// TIA Portal V19 export
FUNCTION_BLOCK "LAF_Checksum"   // FB40, LAD
TITLE = LAF_Checksum / PLC checksum mit ProDiag
AUTHOR : Siemens Digital Industries
FAMILY : LAF
VERSION : 1.2
// The block reads the checksums for PLC standard blocks, for PLC safety blocks and for PLC text lists. The current checksums are compared with the previous values / old values. For each deviation a ProDiag warning is issued, and the colors of the WinCC buttons "Checksum"(SubMenu), "Ok Checksum" and "Settings" (Main Menu) are animated.
// 
// **PLC-Data types**  
// * LAF_typeChecksum  
// * LAF_typeChecksumCatBool  
// * LAF_typeChecksumCatWord  
// 
// **WinCC Screen**  
// 
// {.pageWidth}
// ![Image](LAF_Checksum_PrD/en/image1.PNG)
// 
// **Block call example**  
// {.pageWidth}
// ![Image](LAF_Checksum_PrD/en/image2.PNG)
// The call is shown as “Ladder Diagram” (LAD). 
// 
// **Call interface**  
// The block is called once in the cyclic program. The call takes place in the software unit CentralFunctions -> 05_Diagnostic-> [CallDiagnostic](../Functions/CallDiagnostic.htm)  
// 
// **Internally used “extended instructions / blocks”**  
// GetChecksum, HTA, S_COMP, S_MOVE  
// 
// **Parameters**  
// This block is provided with “pre-defined actual parameters” for structured data types, user constants, system constants etc. Therefor these parameters must be modified only slightly or not at all, if the symbols of DBs, user constants, and system constants have not been changed.
// Der Baustein liest die Checksummen für Standard- und Safety-Bausteine, sowie für Textlisten aus. Die aktuell ausgelesenen Checksummen werden mit den vorherigen Werten (Altwerte) verglichen. Bei Abweichungen wird jeweils eine ProDiag Warnmeldung ausgegeben und die WinCC-Objekte in dem Bild „System & Einstellungen“ farblich animiert. Das Bild ist erreichbar über den Button „System“ (aus jedem Bild, rechts unten).  
// * LSicar_Checksum_PrD:	mit ProDiag-Meldeverfahren 
// * LSicar_Checksum		mit program_Alarm Meldeverfahren
// 
// **PLC-Datentypen**  
//  LSicar_typeChecksum  
//  LSicar_typeChecksumCatBool  
//  LSicar_typeChecksumCatWord  
//  LSicar_typeAlarmText  
//  
// 
// **WinCC-Bild**  
// 
// {.pageWidth}
// ![Image](LSicar_Checksum_PrD/de/image1.PNG)
// 
// **Beispielaufruf**  
// Abbildung in Kontaktplan (KOP), ohne Parameterbeschaltung. D:\Software\Symbols_Icons\BMPs-JPGs-PNGs\Verschiedene\symb_user_goto_transparent.pngEin lauffähiger Programm-Aufruf hierzu ist im „SICAR-StartUp“-Projekt enthalten, incl. der notwendigen HMI-Variablen zur Darstellung der Werte auf dem HMI.  
// 
// **Aufrufschnittstelle**  
// Der Baustein wird einmalig im zyklischen Programm aufgerufen.  
// 
// **Intern verwendete „Erweiterte Anweisungen / Bausteine“**  
// GetChecksum, HTA, S_COMP, S_MOVE  
// 
// **Parameter**
//   
// ![Icon](_Icon/information.PNG) 
// 
// Der Baustein ist mit "Vordefinierten Aktualparametern" versehen für Strukturvariablen, Anwender- und Systemkonstanten etc., die dadurch nicht oder nur geringfügig angepasst werden müssen, vorausgesetzt die Symbolischen Namen von DBs, Anwender-/Systemkonstanten etc. wurden nicht geändert. Die Anpassungen sind notwendig beim Index [i], z.B. für den BA-Bereich oder die HMI-/Panelnummer.  
// 
// * Der Index ist vorbesetzt mit dem Wert [0]. Damit wird auf den Index 0 (Dummy) verwiesen. Sofern der Baustein-Parameter nicht benötigt wird, sind keine Anpassungen notwendig, andernfalls muss der Indexwert angepasst werden.  
// oder  
// * Der Index ist vorbesetzt mit [???]. Dies führt dazu, dass der Aktualparameter beim Bausteinaufruf rot markiert wird; um darauf aufmerksam zu machen, dass der Indexwert des Aktualparameters angepasst werden muss!
// stored: Access Published, IsIECCheckEnabled true, MemoryReserve 100, SetENOAutomatically true
   VAR_INPUT
      plantIdentifier { ExternalAccessible := 'False'; ExternalVisible := 'False'; ExternalWritable := 'False'} : WString[#MAX_CHAR];   // Betriebsmittel Kennzeichen. An diesem Parameter kann ein Text mit max. 24 Zeichen parametriert werden; dies kann beispielweise die Betriebsmittelkennzeichnung sein. Der Wert wird in die ProDiag-Warnmeldung mit eingebracht. / Equipment identifying symbol. The symbol is limited to 24 characters. It can contain the Equipment identifying symbol according to the hardware diagrams. The text assigned here is used for the ProDiag alarm text in the alarm view.
      textListId { ExternalAccessible := 'False'; ExternalVisible := 'False'; ExternalWritable := 'False'} : Int;   // Text list ID
      dateTime { ExternalAccessible := 'False'; ExternalVisible := 'False'; ExternalWritable := 'False'} : Date_And_Time;   // Wird ein Unterschied zwischen der aktuellen und der vorherigen (alten) Checksumme festgestellt, so wird das mit Datum & Uhrzeit abgespeichert und im Bild „Checksumme“ angezeigt. Der Parameter ist vordefiniert und verweist auf nachfolgende Quelle / If the current checksum deviates from the old checksum, date and time are saved and displayed in the screen “Checksum”.
      readChecksum { ExternalAccessible := 'False'; ExternalVisible := 'False'; ExternalWritable := 'False'} : Bool;   // Verwenden Sie hier ein Signal, mit dem die PLC-Checksumme gelesen wird. Es reicht ein Impuls aus. / Assign a signal to read the PLC checksums. A pulse is enough.
      ack { ExternalAccessible := 'False'; ExternalVisible := 'False'; ExternalWritable := 'False'} : Bool;   // Signal mit dem die ProDiag-Warnmeldung quittiert werden kann. Der Parameter ist vordefiniert und verweist auf nachfolgende Quelle. Hinweis: Mit dem globalAck. werden alle anstehenden Meldungen quittiert. Sollen nur die Meldungen für die PLC-Checksumme quittiert werden, so verwenden Sie den Button [OK Checksum] im Bild „Checksum“, siehe WinCC-Bild / For this parameter, assign a signal to reset the ProDiag warnings. Note: All present alarms are reset with the globalAck. If you want to reset only the warnings for the PLC checksums, use the button [OK Checksum] in screen “Checksum".
      hideMessageStandard { ExternalAccessible := 'False'; ExternalVisible := 'False'; ExternalWritable := 'False'} : Bool;   // Der Parameter ist vordefiniert und verweist auf nachfolgende Quelle / The ProDiag warning is suppressed / hidden if a TRUE-Signal is assigned. Note: A TRUE signal does not suppress the color animation of the faceplate and of the WinCC objects in screen “Checksum”. This ensures that the difference of the PLC checksums is visible even if the ProDiag warning is hidden.
      hideMessageSafety { ExternalAccessible := 'False'; ExternalVisible := 'False'; ExternalWritable := 'False'} : Bool;   // Wie bei Parameter „hideMessageStandard“ / Like parameter “hideMessageStandard”
      hideMessageTextlist { ExternalAccessible := 'False'; ExternalVisible := 'False'; ExternalWritable := 'False'} : Bool;   // Wie bei Parameter „hideMessageStandard“ / Like parameter “hideMessageStandard”
   END_VAR
   VAR_OUTPUT
      generalMessage { ExternalAccessible := 'False'; ExternalVisible := 'False'; ExternalWritable := 'False'} : Bool;   // Sammelwarnung / General alarm
   END_VAR
   VAR_IN_OUT
      checksumHmi : "LAF_typeChecksum";   // Transfer of the information for display on the HMI. / PLC checksum for HMI
   END_VAR
   VAR
      statReadChecksumStorage { ExternalAccessible := 'False'; ExternalVisible := 'False'; ExternalWritable := 'False'} : Bool;   // Start: Lesen der PLC Checksummen (Storage) / Start: Read PLC checksum (storage)
      statChecksumStandard { ExternalAccessible := 'False'; ExternalVisible := 'False'; ExternalWritable := 'False'} : Array[0..7] of Byte;   // Checksumme Standard / Checksum Standard
      statChecksumStafety { ExternalAccessible := 'False'; ExternalVisible := 'False'; ExternalWritable := 'False'} : Array[0..7] of Byte;   // Checksumme Safety / Checksum Safety
      statChecksumTextlists { ExternalAccessible := 'False'; ExternalVisible := 'False'; ExternalWritable := 'False'} : Array[0..7] of Byte;   // Checksumme Textlisten / Checksumme Textlists
      statChecksumStandOldNull { ExternalAccessible := 'False'; ExternalVisible := 'False'; ExternalWritable := 'False'} : Bool;   // Vorherige Checksumme = Null (nichts) / Checksum old = null (nothing)
      statChecksumSafeOldNull { ExternalAccessible := 'False'; ExternalVisible := 'False'; ExternalWritable := 'False'} : Bool;   // Vorherige Checksumme = Null (nichts) / Checksum old = null (nothing)
      statChecksumTextlOldNull { ExternalAccessible := 'False'; ExternalVisible := 'False'; ExternalWritable := 'False'} : Bool;   // Vorherige Checksumme = Null (nichts) / Checksum old = null (nothing)
      statChecksumStandDiff { ExternalAccessible := 'False'; ExternalVisible := 'False'; ExternalWritable := 'False'} : Bool;   // Checksumme unterschiedlich Standard / Checksum different Standard
      statChecksumSafeDiff { ExternalAccessible := 'False'; ExternalVisible := 'False'; ExternalWritable := 'False'} : Bool;   // Checksumme unterschiedlich Safety / Checksum different Safety
      statChecksumTextlDiff { ExternalAccessible := 'False'; ExternalVisible := 'False'; ExternalWritable := 'False'} : Bool;   // Checksumme unterschiedlich Textlisten / Checksum different Textlists
      instGetChecksum1 { ExternalAccessible := 'False'; ExternalVisible := 'False'; ExternalWritable := 'False'} : GetChecksum;   // GetChecksum1
      instGetChecksum2 { ExternalAccessible := 'False'; ExternalVisible := 'False'; ExternalWritable := 'False'} : GetChecksum;   // GetChecksum2
      instGetChecksum3 { ExternalAccessible := 'False'; ExternalVisible := 'False'; ExternalWritable := 'False'} : GetChecksum;   // GetChecksum3
      statRetValHta { ExternalAccessible := 'False'; ExternalVisible := 'False'; ExternalWritable := 'False'} : "LAF_typeChecksumCatWord";   // Ret_VAT von HTA / RET_VAL of HTA
      statRisEdgeDiff { ExternalAccessible := 'False'; ExternalVisible := 'False'; ExternalWritable := 'False'} : "LAF_typeChecksumCatBool";   // Steigende Flanke / Rising edge
      statMessageStandModified { ExternalAccessible := 'False'; ExternalVisible := 'False'; ExternalWritable := 'False'} : Bool;   // Meldung: Standard Bausteine wurden modifiziert / Message: Standard blocks are modified
      statMessageSafeModified { ExternalAccessible := 'False'; ExternalVisible := 'False'; ExternalWritable := 'False'} : Bool;   // Meldung: Safety Bausteine wurden modifiziert / Message: Safety blocks are modified
      statMessageTextlModified { ExternalAccessible := 'False'; ExternalVisible := 'False'; ExternalWritable := 'False'} : Bool;   // Meldung: Textlisten wurden modifiziert / Message: Textlists are modified
      statWarnNoStandard { ExternalAccessible := 'False'; ExternalVisible := 'False'; ExternalWritable := 'False'} : UInt;   // Warn Nummer - Standard / Warn number - Standard
      statWarnNoSafety { ExternalAccessible := 'False'; ExternalVisible := 'False'; ExternalWritable := 'False'} : UInt;   // Warn Nummer - Safety / Warn number - Safety
      statWarnNoTextlist { ExternalAccessible := 'False'; ExternalVisible := 'False'; ExternalWritable := 'False'} : UInt;   // Warn Nummer - Textlisten / Warn number - Textlists
   END_VAR
   VAR CONSTANT
      MAX_CHAR : DInt := 24;   // Konstante für Zeichenlänge plantidentifier / Constant length plantidentifier
   END_VAR
   VAR_TEMP   // added for the SCL form of the ladder/FBD networks
      _w1 : Bool;
      _w2 : Bool;
      _w3 : Bool;
   END_VAR
BEGIN

REGION Network 1: Header Info / Änderungshistorie
   // SIEMENS AG / (c)Copyright 2024
   // ------------------------------------------------------------------------------
   // Title:            LAF_InterfaceSignalsBool
   // Comment/Function: The block reads the checksums for PLC standard blocks, for PLC safety blocks and for PLC text lists. The current checksums are compared with the previous values / old values
   // Library/Family:   Library of Automation Framework
   // Author:                Siemens Digital Industry
   // Tested with:       S7-PLCSIM Advanced 6.0
   // Engineering:      TIA Portal V19
   // Restrictions:       ---
   // Requirements:   ---
   // ------------------------------------------------------------------------------
   // Change log table:
   // Version | Date | Expert in charge | Changes applied
   // -------|---------|-------------|--------------------------------------------
   // 01.02.00 | 30.09.2024 | SIMATIC Systems Support | First released version
   // Die Änderungshistorie wird nur in englischer Editiersprache geführt.
END_REGION

REGION Network 2: Description / Beschreibung
   // **Operation mode Automatic / Manual**  
   // The block is independent of operation modes. Therefor it is not assigned to any operation mode area.  
   // 
   // **Alarms**  
   // Alarm texts are stored in the PLC alarm text lists of the software unit GlobalData. This messages are used with proDiag and also in the program alarm version of the block.  
   // 
   // | **No.** | **Message**             |
   // |---------|-------------------------|
   // | 1       | Standard block modified |
   // | 2       | Safety block modified   |
   // | 3       | Textlist modified       |
   // | 4       | Spare4_en               |
   // | 5       | Spare5_en               |
   // | 6       | Spare6_en               |
   // | 7       | Spare7_en               |
   // | 8       | Spare8_en               |
   // 
   // ---
   // 
   // #### PLC Data types 
   // * [LAF_typeChecksum](../Library%20Types/LAF_typeChecksum.htm)  
   // * [LAF_typeChecksumCatBool](../Library%20Types/LAF_typeChecksumCatBool.htm)  
   // * [LAF_typeChecksumCatWord](../Library%20Types/LAF_typeChecksumCatWord.htm)  
   // 
   // 
   // #### WinCC Objects 
   // 
   // **WinCC Screen**  
   // The screen is to be found in the project in the HMI part, in folder “Screens” -> 11_Settings. It consists of several WinCC objects and contains the information shown below.  
   // ![Image](LAF_Checksum_PrD/en/image1.PNG)
   // 
   // ---
   // 
   // #### Further information 
   // 
   // #### Update info
   // 
   // #### Further documentation
   // **Betriebsart Automatik / Hand**  
   // Der Baustein ist keiner Betriebsart / Betriebsartenbereich zugeordnet.  
   // 
   // **Alarme**  
   // Der Baustein generiert die in der PLC-Meldetextliste „PLC_Checksum_PD“ angegebenen Texte als ProDiag-Warnmeldungen, wenn die aktuelle und vorherige (Altwert) Checksumme unterschiedlich sind.  
   // 
   // 
   // Die Textliste „PLC_Checksum_PD“ ist in der PLC-Meldetextliste „GLOBAL_GENERAL_AlarmTextList“ als Eintragsnummer 22 hinterlegt. Siehe auch FB-Parameter: „globalAlarmTextListItem“  
   //  
   // ![Image](LSicar_Checksum_PrD/de/image2.PNG)
   // 
   //  
   // #### PLC Data types 
   // 
   // “_typeChecksum” enthält alle Informationen, die in der Visualisierung angezeigt werden.   
   // 
   // ![Image](LSicar_Checksum_PrD/de/image3.PNG)
   //  
   // “_typeChecksumCatBool” enthält die Struktur für Flankenauswertungen  
   // 
   // ![Image](LSicar_Checksum_PrD/de/image4.PNG)
   //  
   // “_typeChecksumCatWord” enthält die Struktur für RetVal Werte.  
   // 
   // ![Image](LSicar_Checksum_PrD/de/image5.PNG)
   // 
   // Weitere PLC-Datentypen:  
   // 
   // ![Icon](_Icon/reference.PNG)
   // 
   // Siehe LSicar_typeAlarmText.pdf 
   //  
   // 
   // #### WinCC-Bildobjekte
   // 
   // **WinCC-Bild**  
   // Das Bild befindet sich im Projekt im HMI-Teil unter „Bilder“. Es ist erstellt aus mehreren einzelnen WinCC-Objekten und enthält die dargestellten Informationen.  
   // 
   // ![Image](LSicar_Checksum_PrD/de/image6.PNG)
   // 
   // **WinCC-Bildbaustein**  
   // Der Bildbaustein PLC_Checksum befindet sich in der Projektbilbliothek und besteht aus mehreren einzelnen WinCC-Objekten. Er ist in den Startup-Projekten zusätzlich in der Kopfzeile projektiert. Bei Ungleichheit der PLC-Checksummen wird er orange animiert.  
   // In dessen Schnittstelle können Sie die Default-Farbe einstellen. Für das Schnittstellensignal zum Animieren verwenden Sie die HMI-Variable  .summaryModified“.  
   // 
   // ![Image](LSicar_Checksum_PrD/de/image7.PNG)
   // 
   // 
   // #### Further information 
   // 
   // #### Update info
   // 
   // #### Further documentation
END_REGION

REGION Network 3: Call "GetChecksum" and convert to string / Aufruf "GetChecksum" und wandeln in String
   // Read out checksum and convert it to string / Lesen der Prüfsumme und umwandeln in eine Stringvariable
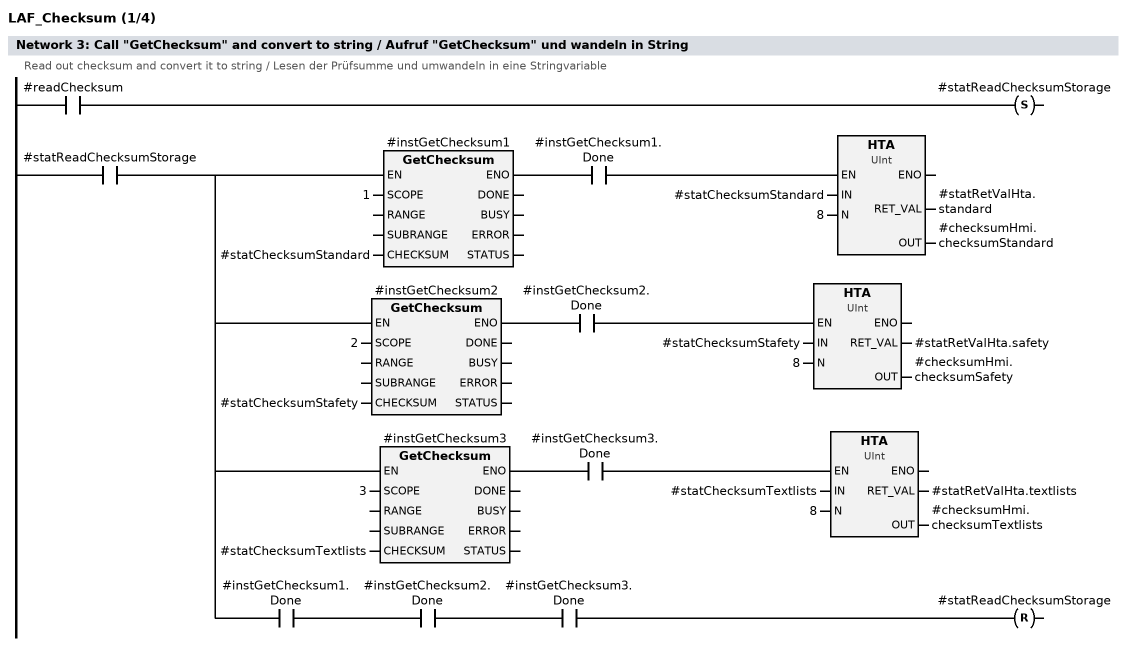
   RUNG wire#powerrail
      Contact( #readChecksum )
      S_Coil( #statReadChecksumStorage )
   END_RUNG
   RUNG wire#powerrail
      Contact( #statReadChecksumStorage )
      wire#w1
      #instGetChecksum1.GetChecksum(Scope := 1, Range :=, Subrange :=, Checksum := #statChecksumStandard, Done =>, Busy =>, Error =>, Status =>)
      Contact( #instGetChecksum1.Done )
      { S7_Templates := "[card := 1, n_type := UInt, in_out_type := Variant]" } HTA(IN := #statChecksumStandard, N := 8, RET_VAL => #statRetValHta.standard, OUT => #checksumHmi.checksumStandard)
   END_RUNG
   RUNG wire#w1
      #instGetChecksum2.GetChecksum(Scope := 2, Range :=, Subrange :=, Checksum := #statChecksumStafety, Done =>, Busy =>, Error =>, Status =>)
      Contact( #instGetChecksum2.Done )
      { S7_Templates := "[card := 1, n_type := UInt, in_out_type := Variant]" } HTA(IN := #statChecksumStafety, N := 8, RET_VAL => #statRetValHta.safety, OUT => #checksumHmi.checksumSafety)
   END_RUNG
   RUNG wire#w1
      #instGetChecksum3.GetChecksum(Scope := 3, Range :=, Subrange :=, Checksum := #statChecksumTextlists, Done =>, Busy =>, Error =>, Status =>)
      Contact( #instGetChecksum3.Done )
      { S7_Templates := "[card := 1, n_type := UInt, in_out_type := Variant]" } HTA(IN := #statChecksumTextlists, N := 8, RET_VAL => #statRetValHta.textlists, OUT => #checksumHmi.checksumTextlists)
   END_RUNG
   RUNG wire#w1
      Contact( #instGetChecksum1.Done )
      Contact( #instGetChecksum2.Done )
      Contact( #instGetChecksum3.Done )
      R_Coil( #statReadChecksumStorage )
   END_RUNG
   // the same network as SCL:
   IF #readChecksum THEN #statReadChecksumStorage := TRUE; END_IF;
   #instGetChecksum1(EN := #statReadChecksumStorage, Scope := 1, Checksum := #statChecksumStandard, ENO => #_w1);   // GetChecksum
   IF #_w1 AND #instGetChecksum1.Done THEN
       #statRetValHta.standard := HTA(IN := #statChecksumStandard, N := 8, OUT => #checksumHmi.checksumStandard);
   END_IF;
   #instGetChecksum2(EN := #statReadChecksumStorage, Scope := 2, Checksum := #statChecksumStafety, ENO => #_w2);   // GetChecksum
   IF #_w2 AND #instGetChecksum2.Done THEN
       #statRetValHta.safety := HTA(IN := #statChecksumStafety, N := 8, OUT => #checksumHmi.checksumSafety);
   END_IF;
   #instGetChecksum3(EN := #statReadChecksumStorage,   // GetChecksum
                     Scope := 3,
                     Checksum := #statChecksumTextlists,
                     ENO => #_w3);
   IF #_w3 AND #instGetChecksum3.Done THEN
       #statRetValHta.textlists := HTA(IN := #statChecksumTextlists, N := 8, OUT => #checksumHmi.checksumTextlists);
   END_IF;
   IF #statReadChecksumStorage AND #instGetChecksum1.Done AND #instGetChecksum2.Done AND #instGetChecksum3.Done THEN
       #statReadChecksumStorage := FALSE;
   END_IF;
END_REGION

REGION Network 4: Overwrite value-before with current-value / Vorheriger Wert mit aktuellem Wert beschreiben
   // Describe old value with current value if old value is still empty (eg. at restart) or if it has been acknowledged with ACK or #HMI.Update_Values_Old / Altwert mit aktuellem Wert beschreiben, falls Altwert noch leer (z.B. bei Neustart) oder wenn Quittiert wurde mit QUIT oder #HMI.Update_Values_Old
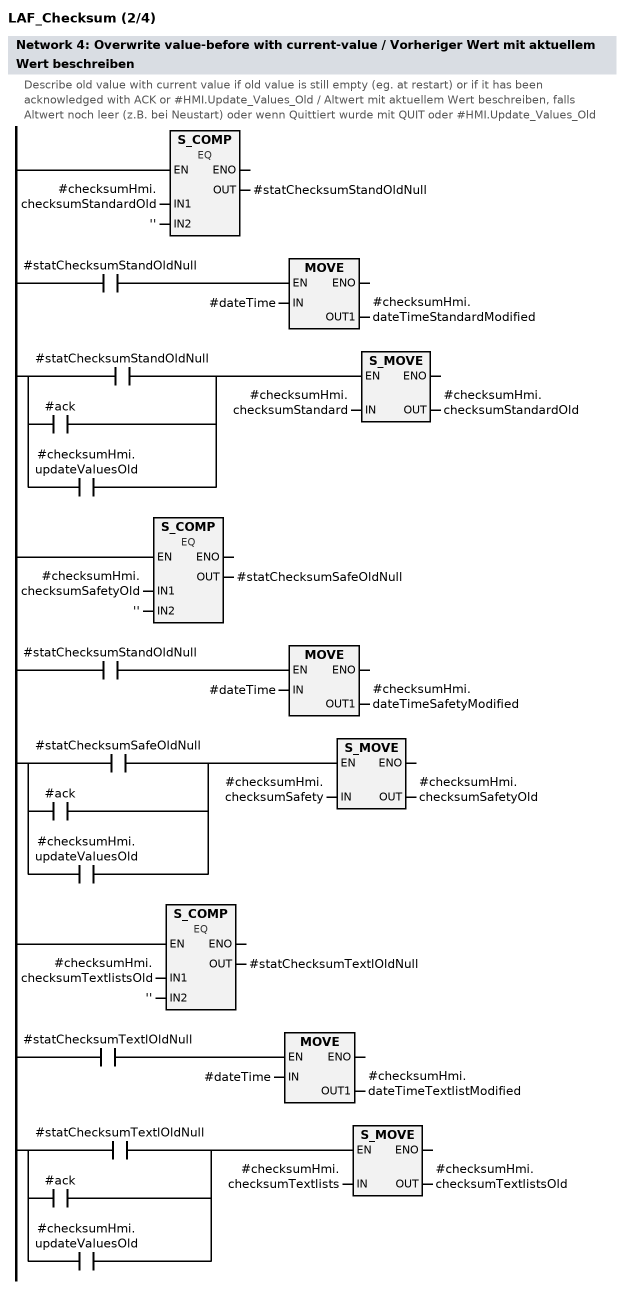
   RUNG wire#powerrail
      { S7_Templates := "[relation := EQ, src_type := String]" } S_COMP(IN1 := #checksumHmi.checksumStandardOld, IN2 := '', OUT => #statChecksumStandOldNull)
   END_RUNG
   RUNG wire#powerrail
      Contact( #statChecksumStandOldNull )
      Move(in := #dateTime, out1 => #checksumHmi.dateTimeStandardModified)
   END_RUNG
   RUNG wire#powerrail
      Contact( #statChecksumStandOldNull )
      wire#w1
      S_Move(in := #checksumHmi.checksumStandard, out => #checksumHmi.checksumStandardOld)
   END_RUNG
   RUNG wire#powerrail
      Contact( #ack )
   END_RUNG wire#w1
   RUNG wire#powerrail
      Contact( #checksumHmi.updateValuesOld )
   END_RUNG wire#w1
   RUNG wire#powerrail
      { S7_Templates := "[relation := EQ, src_type := String]" } S_COMP(IN1 := #checksumHmi.checksumSafetyOld, IN2 := '', OUT => #statChecksumSafeOldNull)
   END_RUNG
   RUNG wire#powerrail
      Contact( #statChecksumStandOldNull )
      Move(in := #dateTime, out1 => #checksumHmi.dateTimeSafetyModified)
   END_RUNG
   RUNG wire#powerrail
      Contact( #statChecksumSafeOldNull )
      wire#w2
      S_Move(in := #checksumHmi.checksumSafety, out => #checksumHmi.checksumSafetyOld)
   END_RUNG
   RUNG wire#powerrail
      Contact( #ack )
   END_RUNG wire#w2
   RUNG wire#powerrail
      Contact( #checksumHmi.updateValuesOld )
   END_RUNG wire#w2
   RUNG wire#powerrail
      { S7_Templates := "[relation := EQ, src_type := String]" } S_COMP(IN1 := #checksumHmi.checksumTextlistsOld, IN2 := '', OUT => #statChecksumTextlOldNull)
   END_RUNG
   RUNG wire#powerrail
      Contact( #statChecksumTextlOldNull )
      Move(in := #dateTime, out1 => #checksumHmi.dateTimeTextlistModified)
   END_RUNG
   RUNG wire#powerrail
      Contact( #statChecksumTextlOldNull )
      wire#w3
      S_Move(in := #checksumHmi.checksumTextlists, out => #checksumHmi.checksumTextlistsOld)
   END_RUNG
   RUNG wire#powerrail
      Contact( #ack )
   END_RUNG wire#w3
   RUNG wire#powerrail
      Contact( #checksumHmi.updateValuesOld )
   END_RUNG wire#w3
   // the same network as SCL:
   S_COMP(IN1 := #checksumHmi.checksumStandardOld, IN2 := '', OUT => #statChecksumStandOldNull);
   IF #statChecksumStandOldNull THEN #checksumHmi.dateTimeStandardModified := #dateTime; END_IF;
   IF #statChecksumStandOldNull OR #ack OR #checksumHmi.updateValuesOld THEN
       #checksumHmi.checksumStandardOld := #checksumHmi.checksumStandard;
   END_IF;
   S_COMP(IN1 := #checksumHmi.checksumSafetyOld, IN2 := '', OUT => #statChecksumSafeOldNull);
   IF #statChecksumStandOldNull THEN #checksumHmi.dateTimeSafetyModified := #dateTime; END_IF;
   IF #statChecksumSafeOldNull OR #ack OR #checksumHmi.updateValuesOld THEN
       #checksumHmi.checksumSafetyOld := #checksumHmi.checksumSafety;
   END_IF;
   S_COMP(IN1 := #checksumHmi.checksumTextlistsOld, IN2 := '', OUT => #statChecksumTextlOldNull);
   IF #statChecksumTextlOldNull THEN #checksumHmi.dateTimeTextlistModified := #dateTime; END_IF;
   IF #statChecksumTextlOldNull OR #ack OR #checksumHmi.updateValuesOld THEN
       #checksumHmi.checksumTextlistsOld := #checksumHmi.checksumTextlists;
   END_IF;
END_REGION

REGION Network 5: Message: Standard blocks are modified / Meldung: Standard Bausteine wurden modifiziert
   // Generate ProDiag message only if it is not deselected (HIDE ... = 0)
   // In the screen always mark the difference in color, by #HMI ... Modified
   // ProDiag-Meldung nur generieren, wenn sie nicht abgewählt ist (HIDE... = 0)
   // Im Bild den Unterschied immer farblich markieren, durch #HMI...Modified
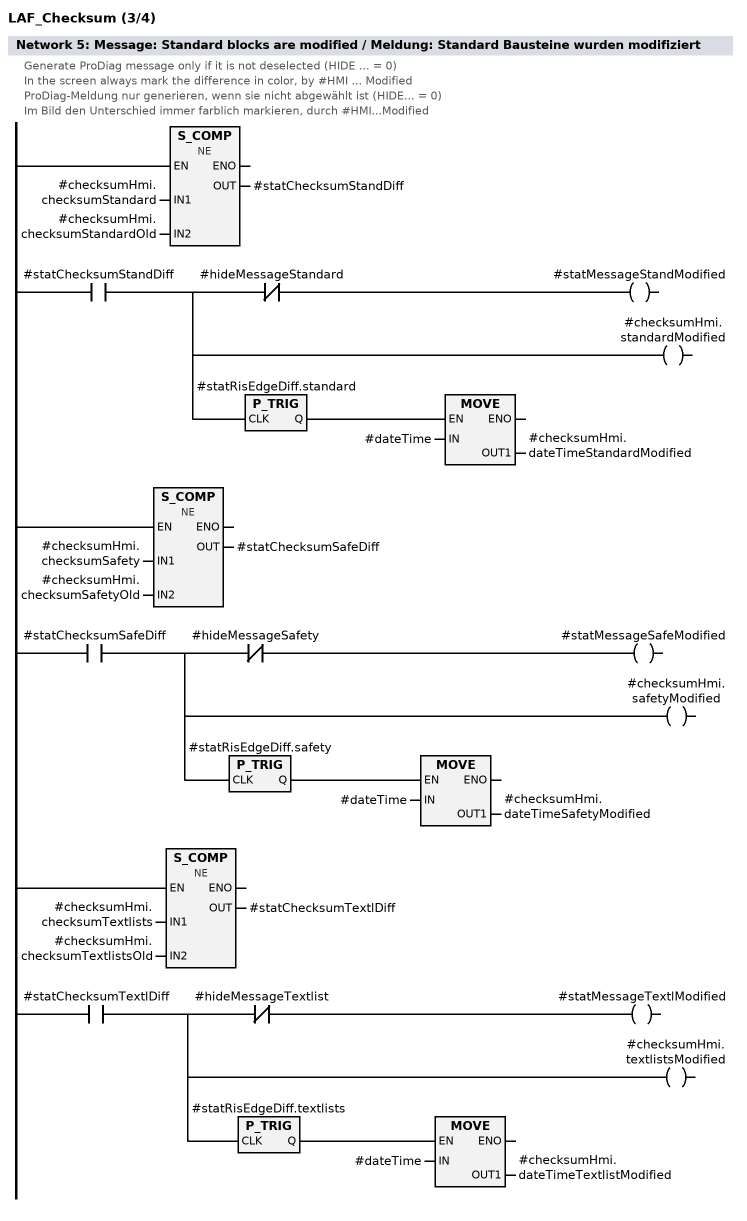
   RUNG wire#powerrail
      { S7_Templates := "[relation := NE, src_type := String]" } S_COMP(IN1 := #checksumHmi.checksumStandard, IN2 := #checksumHmi.checksumStandardOld, OUT => #statChecksumStandDiff)
   END_RUNG
   RUNG wire#powerrail
      Contact( #statChecksumStandDiff )
      wire#w1
      I_Contact( #hideMessageStandard )
      Coil( #statMessageStandModified )
   END_RUNG
   RUNG wire#w1
      Coil( #checksumHmi.standardModified )
   END_RUNG
   RUNG wire#w1
      P_Trig( #statRisEdgeDiff.standard )
      Move(in := #dateTime, out1 => #checksumHmi.dateTimeStandardModified)
   END_RUNG
   RUNG wire#powerrail
      { S7_Templates := "[relation := NE, src_type := String]" } S_COMP(IN1 := #checksumHmi.checksumSafety, IN2 := #checksumHmi.checksumSafetyOld, OUT => #statChecksumSafeDiff)
   END_RUNG
   RUNG wire#powerrail
      Contact( #statChecksumSafeDiff )
      wire#w2
      I_Contact( #hideMessageSafety )
      Coil( #statMessageSafeModified )
   END_RUNG
   RUNG wire#w2
      Coil( #checksumHmi.safetyModified )
   END_RUNG
   RUNG wire#w2
      P_Trig( #statRisEdgeDiff.safety )
      Move(in := #dateTime, out1 => #checksumHmi.dateTimeSafetyModified)
   END_RUNG
   RUNG wire#powerrail
      { S7_Templates := "[relation := NE, src_type := String]" } S_COMP(IN1 := #checksumHmi.checksumTextlists, IN2 := #checksumHmi.checksumTextlistsOld, OUT => #statChecksumTextlDiff)
   END_RUNG
   RUNG wire#powerrail
      Contact( #statChecksumTextlDiff )
      wire#w3
      I_Contact( #hideMessageTextlist )
      Coil( #statMessageTextlModified )
   END_RUNG
   RUNG wire#w3
      Coil( #checksumHmi.textlistsModified )
   END_RUNG
   RUNG wire#w3
      P_Trig( #statRisEdgeDiff.textlists )
      Move(in := #dateTime, out1 => #checksumHmi.dateTimeTextlistModified)
   END_RUNG
   // the same network as SCL:
   S_COMP(IN1 := #checksumHmi.checksumStandard,
          IN2 := #checksumHmi.checksumStandardOld,
          OUT => #statChecksumStandDiff);
   #statMessageStandModified := #statChecksumStandDiff AND NOT #hideMessageStandard;
   #checksumHmi.standardModified := #statChecksumStandDiff;
   #_w1 := #statChecksumStandDiff AND NOT #statRisEdgeDiff.standard;   // rising edge
   #statRisEdgeDiff.standard := #statChecksumStandDiff;
   IF #_w1 THEN #checksumHmi.dateTimeStandardModified := #dateTime; END_IF;
   S_COMP(IN1 := #checksumHmi.checksumSafety,
          IN2 := #checksumHmi.checksumSafetyOld,
          OUT => #statChecksumSafeDiff);
   #statMessageSafeModified := #statChecksumSafeDiff AND NOT #hideMessageSafety;
   #checksumHmi.safetyModified := #statChecksumSafeDiff;
   #_w2 := #statChecksumSafeDiff AND NOT #statRisEdgeDiff.safety;   // rising edge
   #statRisEdgeDiff.safety := #statChecksumSafeDiff;
   IF #_w2 THEN #checksumHmi.dateTimeSafetyModified := #dateTime; END_IF;
   S_COMP(IN1 := #checksumHmi.checksumTextlists,
          IN2 := #checksumHmi.checksumTextlistsOld,
          OUT => #statChecksumTextlDiff);
   #statMessageTextlModified := #statChecksumTextlDiff AND NOT #hideMessageTextlist;
   #checksumHmi.textlistsModified := #statChecksumTextlDiff;
   #_w3 := #statChecksumTextlDiff AND NOT #statRisEdgeDiff.textlists;   // rising edge
   #statRisEdgeDiff.textlists := #statChecksumTextlDiff;
   IF #_w3 THEN #checksumHmi.dateTimeTextlistModified := #dateTime; END_IF;
END_REGION

REGION Network 6: General messages / Sammelmeldungen
   // Generate message if checksum is changed / Erstellen einer Meldung wenn die Prüfsumme geänder wird
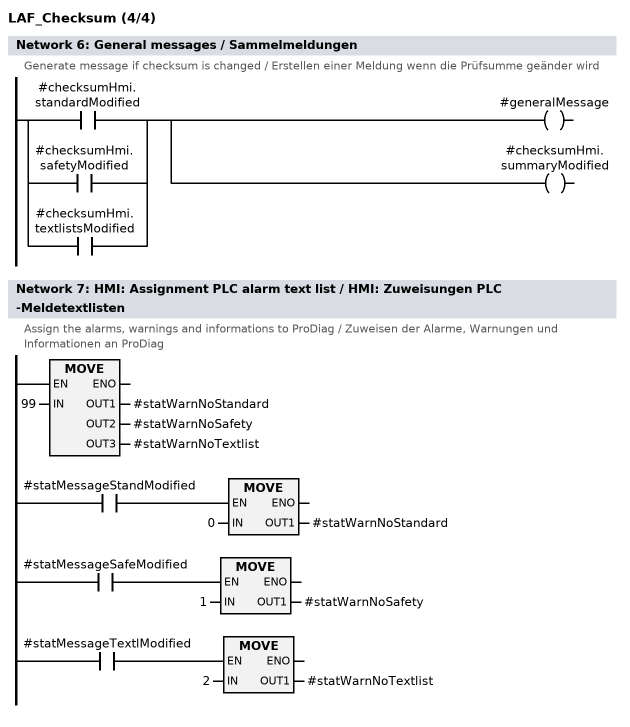
   RUNG wire#powerrail
      Contact( #checksumHmi.standardModified )
      wire#w1
      Coil( #generalMessage )
   END_RUNG
   RUNG wire#powerrail
      Contact( #checksumHmi.safetyModified )
   END_RUNG wire#w1
   RUNG wire#powerrail
      Contact( #checksumHmi.textlistsModified )
   END_RUNG wire#w1
   RUNG wire#w1
      Coil( #checksumHmi.summaryModified )
   END_RUNG
   // the same network as SCL:
   #generalMessage := #checksumHmi.standardModified OR #checksumHmi.safetyModified OR #checksumHmi.textlistsModified;
   #checksumHmi.summaryModified := #generalMessage;
END_REGION

REGION Network 7: HMI: Assignment PLC alarm text list / HMI: Zuweisungen PLC -Meldetextlisten
   // Assign the alarms, warnings and informations to ProDiag / Zuweisen der Alarme, Warnungen und Informationen an ProDiag
   RUNG wire#powerrail
      Move(in := 99, out1 => #statWarnNoStandard, out2 => #statWarnNoSafety, out3 => #statWarnNoTextlist)
   END_RUNG
   RUNG wire#powerrail
      Contact( #statMessageStandModified )
      Move(in := 0, out1 => #statWarnNoStandard)
   END_RUNG
   RUNG wire#powerrail
      Contact( #statMessageSafeModified )
      Move(in := 1, out1 => #statWarnNoSafety)
   END_RUNG
   RUNG wire#powerrail
      Contact( #statMessageTextlModified )
      Move(in := 2, out1 => #statWarnNoTextlist)
   END_RUNG
   // the same network as SCL:
   #statWarnNoStandard := 99;
   #statWarnNoSafety := 99;
   #statWarnNoTextlist := 99;
   IF #statMessageStandModified THEN #statWarnNoStandard := 0; END_IF;
   IF #statMessageSafeModified THEN #statWarnNoSafety := 1; END_IF;
   IF #statMessageTextlModified THEN #statWarnNoTextlist := 2; END_IF;
END_REGION
END_FUNCTION_BLOCK
